(* PLC project dcmotor, Dassault Systèmes ControlBuild 2024x Refresh1 *)
(* stored: creationDateTime 2024-03-13T11:33:32-01:00 *)

FUNCTION_BLOCK stimuli_model
  VAR_OUTPUT
    U : REAL := 0.0;
    M_load : REAL := 0.0;
  END_VAR


ACTION C_source_code:

END_ACTION
END_FUNCTION_BLOCK

FUNCTION_BLOCK edrive_mass
  VAR_INPUT
    M_A : REAL := 0.0;
    M_B : REAL := 0.0;
  END_VAR
  VAR_OUTPUT
    phiA : REAL := 0.0;
    wB : REAL := 0.0;
    wA : REAL := 0.0;
    phiB : REAL := 0.0;
  END_VAR


ACTION C_source_code:

END_ACTION
END_FUNCTION_BLOCK

FUNCTION_BLOCK emachine_model
  VAR_INPUT
    phi : REAL := 0.0;
    w : REAL := 0.0;
    U : REAL := 0.0;
  END_VAR
  VAR_OUTPUT
    M : REAL := 0.0;
    I : REAL := 0.0;
  END_VAR


ACTION C_source_code:

END_ACTION
END_FUNCTION_BLOCK

PROGRAM sut
  VAR_INPUT
    M_load : REAL := 0.0;
    U : REAL := 0.0;
  END_VAR
  VAR_OUTPUT
    I : REAL := 0.0;
    wB : REAL := 0.0;
    M_mot : REAL := 0.0;
    phiB : REAL := 0.0;
  END_VAR

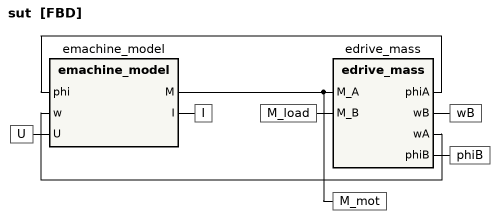
(* FBD diagram, written out as Structured Text *)
edrive_mass(M_A := emachine_model.M, M_B := M_load);
emachine_model(phi := edrive_mass.phiA, w := edrive_mass.wA, U := U);
M_mot := emachine_model.M;
wB := edrive_mass.wB;
I := emachine_model.I;
phiB := edrive_mass.phiB;
END_PROGRAM

PROGRAM my_app.dcmotor
  VAR_OUTPUT
    wB : REAL := 0.0;
    I : REAL := 0.0;
    U : REAL := 0.0;
    M_mot : REAL := 0.0;
  END_VAR

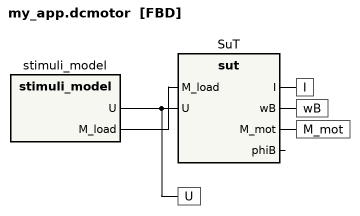
(* FBD diagram, written out as Structured Text *)
stimuli_model();
SuT(M_load := stimuli_model.M_load, U := stimuli_model.U);
I := SuT.I;
wB := SuT.wB;
M_mot := SuT.M_mot;
U := stimuli_model.U;
END_PROGRAM
